(* IEC 61131-3 sources: Industry-PLC-LLM/data/PLCBEAD_repo/PLCBEAD_PLCEmbed-main/PLC-BEAD/Source/GEB/DAY_TO_TIME, 1 file *)

(* ---- DAY_TO_TIME.ST ---- *)
FUNCTION DAY_TO_TIME:TIME
	VAR_INPUT
		IN :	REAL;
	END_VAR

	DAY_TO_TIME := DINT_TO_TIME(UDINT_TO_DINT(_REAL_TO_UDINT(IN * REAL#86400000.00)));
END_FUNCTION

FUNCTION _REAL_TO_UDINT:UDINT
  VAR_INPUT
    X :	REAL;
  END_VAR

  IF REAL_TO_UDINT(0.5) = UDINT#1 THEN
    _REAL_TO_UDINT := REAL_TO_UDINT(X);
  ELSIF X > 0.0 THEN
    _REAL_TO_UDINT := REAL_TO_UDINT(X+0.5);
  ELSIF X < 0.0 THEN
    _REAL_TO_UDINT := REAL_TO_UDINT(X-0.5);
  ELSE
    _REAL_TO_UDINT := UDINT#0;
  END_IF;
END_FUNCTION

PROGRAM program0
  VAR
    LocalVar0 : REAL;
	LocalOUT  : TIME;
  END_VAR
  	LocalOUT := DAY_TO_TIME(LocalVar0);
END_PROGRAM
